{attribute 'qualified_only'}
{attribute 'strict'}
TYPE E_LSPM_LiftType :
(
	E_UNKNOWN,
	E_ENCODER,
	E_INDUCTIVE_SENSORS
);
END_TYPE

(* stored: Version 1.1.0.1, ProductVersion 3.1.4024.4
   DUT E_LSPM_LiftType: Id {897fa2fa-60e1-4f62-b968-6207945b2b9e} *)
